FUNCTION_BLOCK ABSTRACT CyclicBase IMPLEMENTS ICyclic
VAR
END_VAR

METHOD PUBLIC ABSTRACT Cycle : BOOL
VAR_INPUT
END_VAR
END_METHOD

END_FUNCTION_BLOCK

(* stored: Version 1.1.0.1, ProductVersion 3.1.4024.12
   POU CyclicBase: Id {99312e67-14c0-45fd-9386-851ad24e0c0b}, SpecialFunc None
   Method Cycle: Id {2c231b79-b18c-464a-8764-d74ad790a470} *)
